// TIA Portal project "Al Qasim" (V16)

(* hardware
DEVICE "S7-1200 station_1"  S7-1200 Station
   slot 0: "Rack_0"  S7-1200 Rack  Rack  V1.0
   slot 1: "George"  CPU 1212C AC/DC/Rly  6ES7 212-1BE40-0XB0  V4.3
   slot 2: "DI 16x24VDC_1"  6ES7 221-1BF32-0XB0  V2.0
   slot 3: "CB 1241 (RS485)"  CB 1241 (RS485)  6ES7 241-1CH30-1XB0  V1.0
*)

// ===== PLC "George"  CPU 1212C AC/DC/Rly =====

VAR_GLOBAL   // PLC tag table "Default tag table"
   "System_Byte" AT %MB1000 : Byte;
   "FirstScan" AT %M1000.0 : Bool;
   "DiagStatusUpdate" AT %M1000.1 : Bool;
   "AlwaysTRUE" AT %M1000.2 : Bool;
   "AlwaysFALSE" AT %M1000.3 : Bool;
   "Clock_Byte" AT %MB1001 : Byte;
   "Clock_10Hz" AT %M1001.0 : Bool;
   "Clock_5Hz" AT %M1001.1 : Bool;
   "Clock_2.5Hz" AT %M1001.2 : Bool;
   "Clock_2Hz" AT %M1001.3 : Bool;
   "Clock_1.25Hz" AT %M1001.4 : Bool;
   "Clock_1Hz" AT %M1001.5 : Bool;
   "Clock_0.625Hz" AT %M1001.6 : Bool;
   "Clock_0.5Hz" AT %M1001.7 : Bool;
   "TS in Progress" AT %M0.0 : Bool;
   "TS Complete" AT %M0.1 : Bool;
   "initial switch ok" AT %M0.2 : Bool;
   "Datalog pulse" AT %M0.4 : Bool;
   "save name" AT %MB3 : Char;
   "allow datalogging" AT %M0.5 : Bool;
END_VAR

VAR_GLOBAL   // PLC tag table "Inputs"
   "Master Overide" AT %I0.0 : Bool;
   "Overide Pump 1" AT %I0.1 : Bool;
   "Overide Pump 2" AT %I0.2 : Bool;
   "Overide Pump 3" AT %I0.3 : Bool;
   "Overide Pump 4" AT %I0.4 : Bool;
   "Overide Pump 5" AT %I0.5 : Bool;
   "Float Inlet" AT %I0.6 : Bool;
   "Float Outlet" AT %I0.7 : Bool;
   "Float Stage" AT %I1.0 : Bool;
   "PB_Start" AT %I1.1 : Bool;
   "PB_Stop" AT %I1.2 : Bool;
END_VAR

VAR_GLOBAL   // PLC tag table "Outputs"
   "Pump 1" AT %Q0.0 : Bool;
   "Pump 2" AT %Q0.1 : Bool;
   "Pump 3" AT %Q0.2 : Bool;
   "Pump 4" AT %Q0.3 : Bool;
   "Pump 5" AT %Q0.4 : Bool;
   "Prog is running" AT %Q0.5 : Bool;
END_VAR

VAR_GLOBAL   // PLC tag table "Memory"
   "Main Function Loop" AT %MW1 : Int;   // 0= start up, 1 = stop, 2 = go, =3 Master Control
   "Run Mode" AT %MW4 : Int;   // 0 = Normal running, 1= tank switch, 2 inverted Humidity error
   "Tank Switch Mode Bit" AT %MW6 : Int;
   "OK to Switch" AT %M8.0 : Bool;
   "addy" AT %MW10 : Int;
   "Start a datalog session" AT %M0.3 : Bool;
   "logging ID" AT %MD12 : DInt;
   "OS log reset" AT %M0.6 : Bool;
   "OS1" AT %M0.7 : Bool;
END_VAR

VAR_GLOBAL   // PLC tag table "Retained memory"
   "Namer Logger" AT %MD1 : DInt;
   "name logger 2" AT %MD16 : DInt;
END_VAR

DATA_BLOCK "Stop_DB"   // DB1
{ S7_Optimized_Access := 'TRUE' }
VERSION : 0.1
// stored: InstanceOfName Stop
"Stop"
BEGIN
END_DATA_BLOCK

DATA_BLOCK "Auto Run_DB"   // DB2
{ S7_Optimized_Access := 'TRUE' }
VERSION : 0.1
// stored: InstanceOfName Auto Run
"Auto Run"
BEGIN
END_DATA_BLOCK

DATA_BLOCK "Manual Control_DB"   // DB9
{ S7_Optimized_Access := 'TRUE' }
VERSION : 0.1
// stored: InstanceOfName Manual Control
"Manual Control"
BEGIN
END_DATA_BLOCK

DATA_BLOCK "Modbus_DB"   // DB14
{ S7_Optimized_Access := 'TRUE' }
VERSION : 0.1
// stored: InstanceOfName Modbus
"Modbus"
BEGIN
END_DATA_BLOCK

DATA_BLOCK "Data process_DB"   // DB15
{ S7_Optimized_Access := 'TRUE' }
VERSION : 0.1
// stored: InstanceOfName Data process
"Data process"
BEGIN
END_DATA_BLOCK

// folder: Data

DATA_BLOCK "Data"   // DB3
{ S7_Optimized_Access := 'TRUE' }
VERSION : 0.1
   VAR
      "Inside Humidity" : Real := 80.0;
      "Inside Temp" : Real := 20.0;
      "Outside Humidity" : Real := 20.0;
      "Outside Temp" : Real := 30.0;
      "Temp Set Point" : Real := 18.0;
      "Hum Diff Set Point" : Real := 5.0;
      "Reset Timer" : Time := T#60s;
      "Tank Switch in progress" : Real;   // When Tank is switching, value is 100
      "Min Humidity" : Real := 40.0;   // Min humidity coming off the pad
   END_VAR
BEGIN
END_DATA_BLOCK

DATA_BLOCK "Modbus Data"   // DB13
{ S7_Optimized_Access := 'FALSE' }
VERSION : 0.1
   VAR
      "H&T" : Array[0..1] of Int;
      "Modbus Busy" : Bool;
   END_VAR
BEGIN
END_DATA_BLOCK

// folder: Data/Data Logging

DATA_BLOCK "Data Logging Config"   // DB21
{ S7_Optimized_Access := 'TRUE' }
VERSION : 0.1
   VAR
      "Name" : String := 'ash';
      ID : DInt := 0;
      Hedder : String := 'Ambient Temp,Ambient Hum,Inside Temp,Inside Hum,Tank Switch In Progress';
      "Data Log Data" : Struct
         "Data to be logged" : Array[0..4] of Real;
      END_STRUCT;
      "Start Done" : Bool;
      "Memory Allocation" : DInt := 5000;
      "Datalog Time Interval" : Time := T#1S;
   END_VAR
BEGIN
END_DATA_BLOCK

DATA_BLOCK "Create Data Log_DB"   // DB22
{ S7_Optimized_Access := 'TRUE' }
VERSION : 0.1
// stored: InstanceOfName Create Data Log
"Create Data Log"
BEGIN
END_DATA_BLOCK

// folder: Program Modes

DATA_BLOCK "Normal Running_DB"   // DB4
{ S7_Optimized_Access := 'TRUE' }
VERSION : 0.1
// stored: InstanceOfName Normal Running
"Normal Running"
BEGIN
END_DATA_BLOCK

DATA_BLOCK "Tank Switch_DB"   // DB5
{ S7_Optimized_Access := 'TRUE' }
VERSION : 0.1
// stored: InstanceOfName Tank Switch
"Tank Switch"
BEGIN
END_DATA_BLOCK

DATA_BLOCK "Tank Switch_DB_1"   // DB7
{ S7_Optimized_Access := 'TRUE' }
VERSION : 0.1
// stored: InstanceOfName Tank Switch
"Tank Switch"
BEGIN
END_DATA_BLOCK

DATA_BLOCK "Stop_DB_1"   // DB8
{ S7_Optimized_Access := 'TRUE' }
VERSION : 0.1
// stored: InstanceOfName Stop
"Stop"
BEGIN
END_DATA_BLOCK

DATA_BLOCK "Normal Running_DB_1"   // DB17
{ S7_Optimized_Access := 'TRUE' }
VERSION : 0.1
// stored: InstanceOfName Normal Running
"Normal Running"
BEGIN
END_DATA_BLOCK

DATA_BLOCK "Data Logging_DB"   // DB25
{ S7_Optimized_Access := 'TRUE' }
VERSION : 0.1
// stored: InstanceOfName Data Logging
"Data Logging"
BEGIN
END_DATA_BLOCK

// folder: System blocks/Program resources

DATA_BLOCK "IEC_Timer_0_DB"   // DB6
{ S7_Optimized_Access := 'TRUE' }
AUTHOR : Simatic
FAMILY : IEC
NAME : IEC_TMR
VERSION : 1.0
// stored: InstanceOfName IEC_TIMER
"IEC_TIMER"
BEGIN
END_DATA_BLOCK

DATA_BLOCK "IEC_Timer_0_DB_2"   // DB11
{ S7_Optimized_Access := 'TRUE' }
AUTHOR : Simatic
FAMILY : IEC
NAME : IEC_TMR
VERSION : 1.0
// stored: InstanceOfName IEC_TIMER
"IEC_TIMER"
BEGIN
END_DATA_BLOCK

DATA_BLOCK "IEC_Timer_0_DB_3"   // DB16
{ S7_Optimized_Access := 'TRUE' }
AUTHOR : Simatic
FAMILY : IEC
NAME : IEC_TMR
VERSION : 1.0
// stored: InstanceOfName IEC_TIMER
"IEC_TIMER"
BEGIN
END_DATA_BLOCK

DATA_BLOCK "IEC_Timer_0_DB_1"   // DB24
{ S7_Optimized_Access := 'TRUE' }
AUTHOR : Simatic
FAMILY : IEC
NAME : IEC_TMR
VERSION : 1.0
// stored: InstanceOfName IEC_TIMER
"IEC_TIMER"
BEGIN
END_DATA_BLOCK

// folder: (top level)

FUNCTION_BLOCK "Modbus"   // FB6, LAD
{ S7_Optimized_Access := 'TRUE' }
VERSION : 0.1
BEGIN

REGION Network 1: To read T&H from 2 sensors @ address 2 and 3
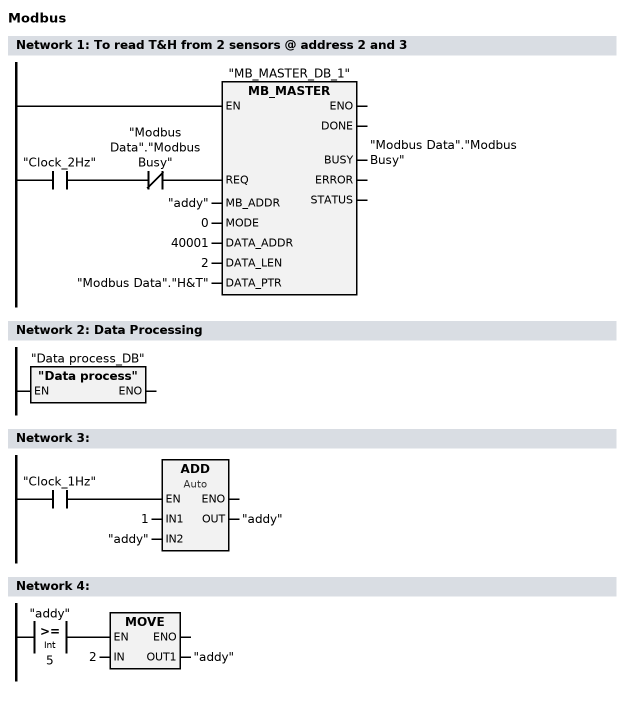
   "MB_MASTER_DB_1"(REQ := "Clock_2Hz" AND NOT "Modbus Data"."Modbus Busy",   // MB_MASTER
                    MB_ADDR := "addy",
                    MODE := 0,
                    DATA_ADDR := 40001,
                    DATA_LEN := 2,
                    DATA_PTR := "Modbus Data"."H&T",
                    BUSY => "Modbus Data"."Modbus Busy");
END_REGION

REGION Network 2: Data Processing
   RUNG wire#powerrail
      "Data process_DB"()
   END_RUNG
   // the same network as SCL:
   "Data process_DB"();   // "Data process"
END_REGION

REGION Network 3
   RUNG wire#powerrail
      Contact( "Clock_1Hz" )
      Add(in1 := 1, in2 := "addy", out => "addy")
   END_RUNG
   // the same network as SCL:
   IF "Clock_1Hz" THEN "addy" := 1 + "addy"; END_IF;
END_REGION

REGION Network 4
   RUNG wire#powerrail
      { S7_Templates := "SrcType := Int" } GE_Contact(in1 := "addy", in2 := 5)
      Move(in := 2, out1 => "addy")
   END_RUNG
   // the same network as SCL:
   IF "addy" >= 5 THEN "addy" := 2; END_IF;
END_REGION
END_FUNCTION_BLOCK

ORGANIZATION_BLOCK "Main"   // OB1, LAD, ProgramCycle
TITLE = "Main Program Sweep (Cycle)"
{ S7_Optimized_Access := 'TRUE' }
VERSION : 0.1
   VAR_INPUT
      Initial_Call : Bool;   // Initial call of this OB
      Remanence : Bool;   // =True, if remanent data are available
   END_VAR
   VAR_TEMP   // added for the SCL form of the ladder/FBD networks
      _w1 : Bool;
      _w2 : Bool;
   END_VAR
BEGIN

REGION Network 1: Select Main function Loop
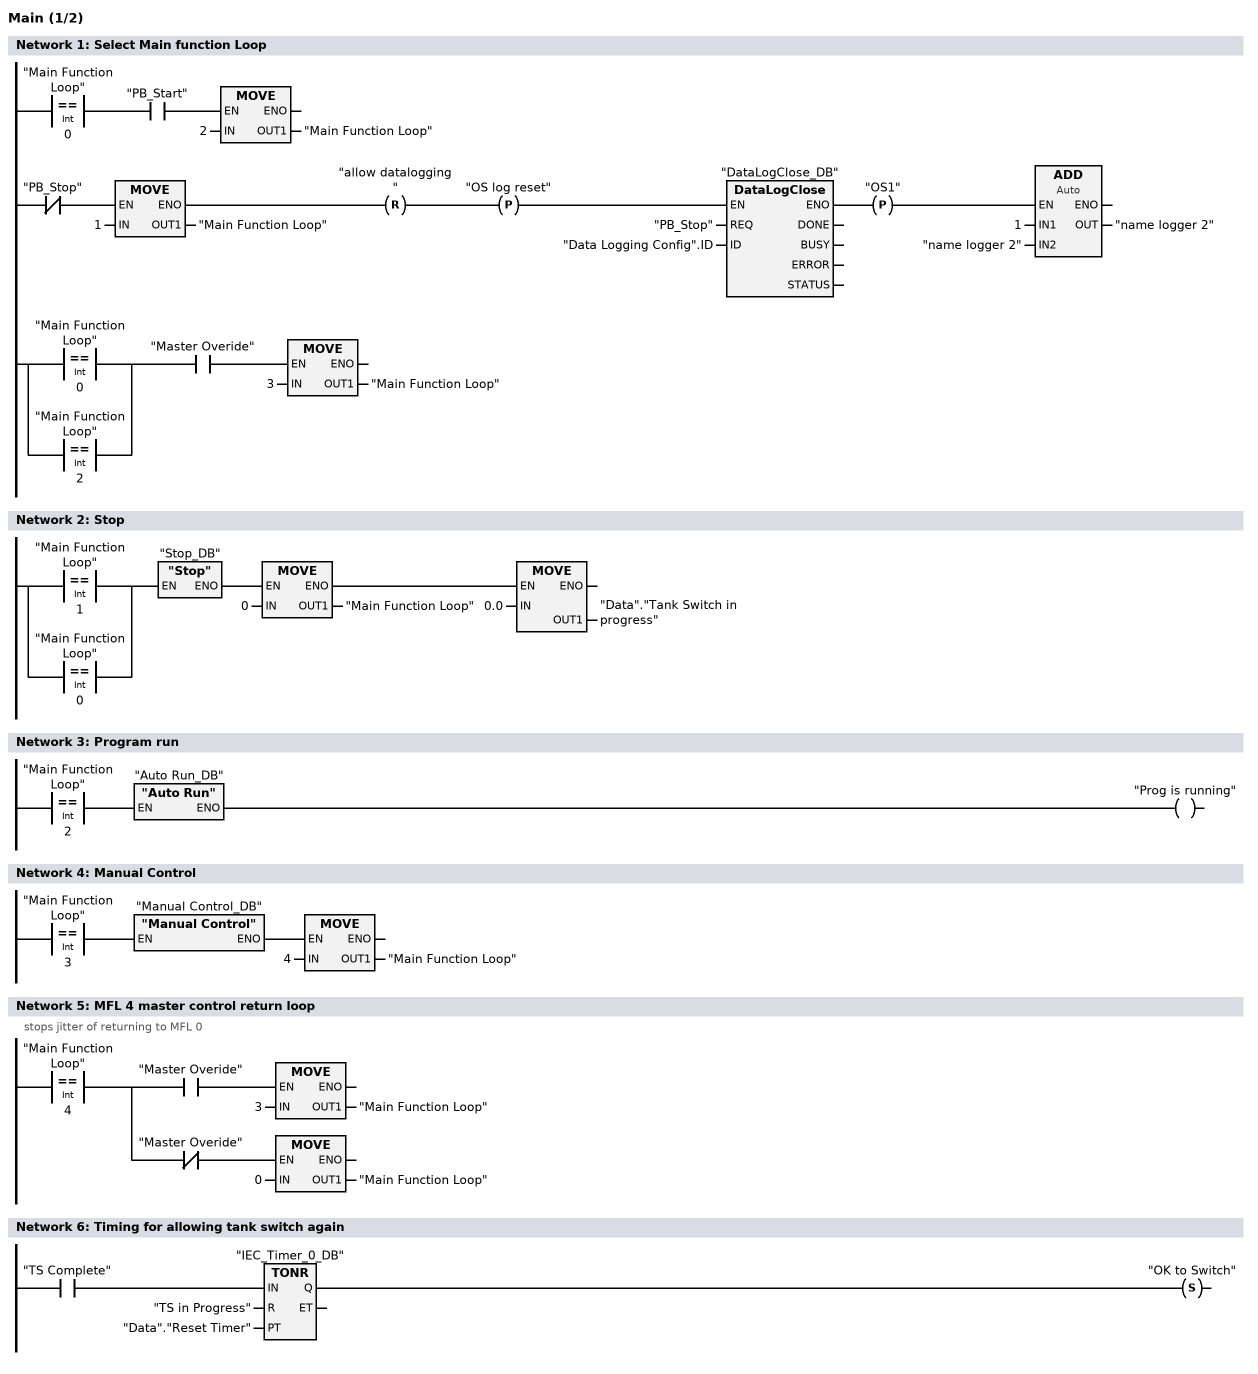
   // ENO of a box is taken as its EN; it also drops when the box reports an error
   IF ("Main Function Loop" = 0) AND "PB_Start" THEN "Main Function Loop" := 2; END_IF;
   IF NOT "PB_Stop" THEN
       "Main Function Loop" := 1;
       "allow datalogging" := FALSE;
   END_IF;
   #_w1 := NOT "PB_Stop" AND NOT "OS log reset";   // rising edge
   "OS log reset" := NOT "PB_Stop";
   IF #_w1 THEN
       "DataLogClose_DB"(REQ := "PB_Stop", ID := "Data Logging Config".ID);   // DataLogClose
   END_IF;
   #_w2 := #_w1 AND NOT "OS1";   // rising edge
   "OS1" := #_w1;
   IF #_w2 THEN "name logger 2" := 1 + "name logger 2"; END_IF;
   IF (("Main Function Loop" = 0) OR ("Main Function Loop" = 2)) AND "Master Overide" THEN
       "Main Function Loop" := 3;
   END_IF;
END_REGION

REGION Network 2: Stop
   RUNG wire#powerrail
      { S7_Templates := "SrcType := Int" } EQ_Contact(in1 := "Main Function Loop", in2 := 1)
      wire#w1
      "Stop_DB"()
      Move(in := 0, out1 => "Main Function Loop")
      Move(in := 0.0, out1 => "Data"."Tank Switch in progress")
   END_RUNG
   RUNG wire#powerrail
      { S7_Templates := "SrcType := Int" } EQ_Contact(in1 := "Main Function Loop", in2 := 0)
   END_RUNG wire#w1
   // the same network as SCL:
   "Stop_DB"(EN := ("Main Function Loop" = 1) OR ("Main Function Loop" = 0), ENO => #_w1);   // "Stop"
   IF #_w1 THEN
       "Main Function Loop" := 0;
       "Data"."Tank Switch in progress" := 0.0;
   END_IF;
END_REGION

REGION Network 3: Program run
   RUNG wire#powerrail
      { S7_Templates := "SrcType := Int" } EQ_Contact(in1 := "Main Function Loop", in2 := 2)
      "Auto Run_DB"()
      Coil( "Prog is running" )
   END_RUNG
   // the same network as SCL:
   "Auto Run_DB"(EN := "Main Function Loop" = 2, ENO => #_w1);   // "Auto Run"
   "Prog is running" := #_w1;
END_REGION

REGION Network 4: Manual Control
   RUNG wire#powerrail
      { S7_Templates := "SrcType := Int" } EQ_Contact(in1 := "Main Function Loop", in2 := 3)
      "Manual Control_DB"()
      Move(in := 4, out1 => "Main Function Loop")
   END_RUNG
   // the same network as SCL:
   "Manual Control_DB"(EN := "Main Function Loop" = 3, ENO => #_w1);   // "Manual Control"
   IF #_w1 THEN "Main Function Loop" := 4; END_IF;
END_REGION

REGION Network 5: MFL 4 master control return loop
   // stops jitter of returning to MFL 0
   RUNG wire#powerrail
      { S7_Templates := "SrcType := Int" } EQ_Contact(in1 := "Main Function Loop", in2 := 4)
      wire#w1
      Contact( "Master Overide" )
      Move(in := 3, out1 => "Main Function Loop")
   END_RUNG
   RUNG wire#w1
      I_Contact( "Master Overide" )
      Move(in := 0, out1 => "Main Function Loop")
   END_RUNG
   // the same network as SCL:
   #_w1 := "Main Function Loop" = 4;
   IF #_w1 AND "Master Overide" THEN "Main Function Loop" := 3; END_IF;
   IF #_w1 AND NOT "Master Overide" THEN "Main Function Loop" := 0; END_IF;
END_REGION

REGION Network 6: Timing for allowing tank switch again
   "IEC_Timer_0_DB".TONR(IN := "TS Complete", R := "TS in Progress", PT := "Data"."Reset Timer");
   IF "IEC_Timer_0_DB".Q THEN "OK to Switch" := TRUE; END_IF;
END_REGION

REGION Network 7: reset easter egg (hold stop for 5 sec)
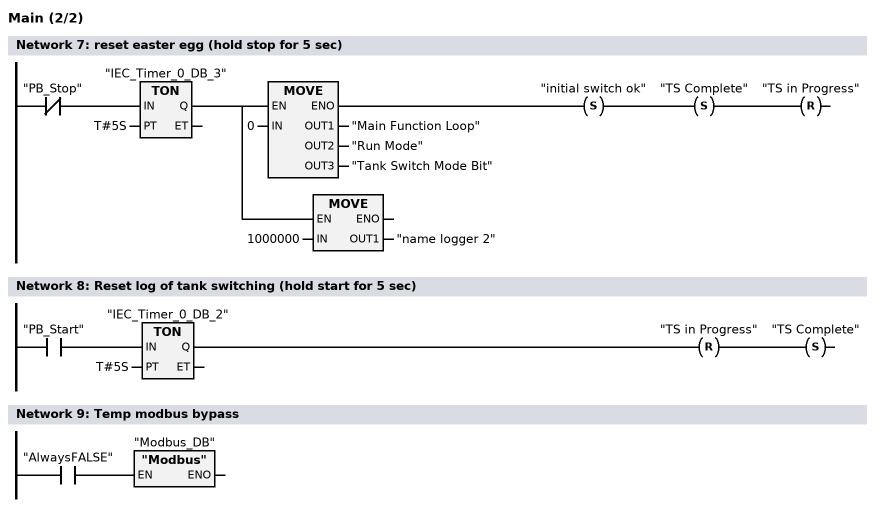
   "IEC_Timer_0_DB_3".TON(IN := NOT "PB_Stop", PT := T#5S);
   IF "IEC_Timer_0_DB_3".Q THEN
       "Main Function Loop" := 0;
       "Run Mode" := 0;
       "Tank Switch Mode Bit" := 0;
       "initial switch ok" := TRUE;
       "TS Complete" := TRUE;
       "TS in Progress" := FALSE;
       "name logger 2" := 1000000;
   END_IF;
END_REGION

REGION Network 8: Reset log of tank switching (hold start for 5 sec)
   "IEC_Timer_0_DB_2".TON(IN := "PB_Start", PT := T#5S);
   IF "IEC_Timer_0_DB_2".Q THEN
       "TS in Progress" := FALSE;
       "TS Complete" := TRUE;
   END_IF;
END_REGION

REGION Network 9: Temp modbus bypass
   RUNG wire#powerrail
      Contact( "AlwaysFALSE" )
      "Modbus_DB"()
   END_RUNG
   // the same network as SCL:
   IF "AlwaysFALSE" THEN
       "Modbus_DB"();   // "Modbus"
   END_IF;
END_REGION
END_ORGANIZATION_BLOCK

ORGANIZATION_BLOCK "Startup"   // OB100, LAD, Startup
TITLE = "Complete Restart"
{ S7_Optimized_Access := 'TRUE' }
VERSION : 0.1
   VAR_INPUT
      LostRetentive : Bool;   // True if retentive data are lost
      LostRTC : Bool;   // True if date and time are lost
   END_VAR
BEGIN

REGION Network 1
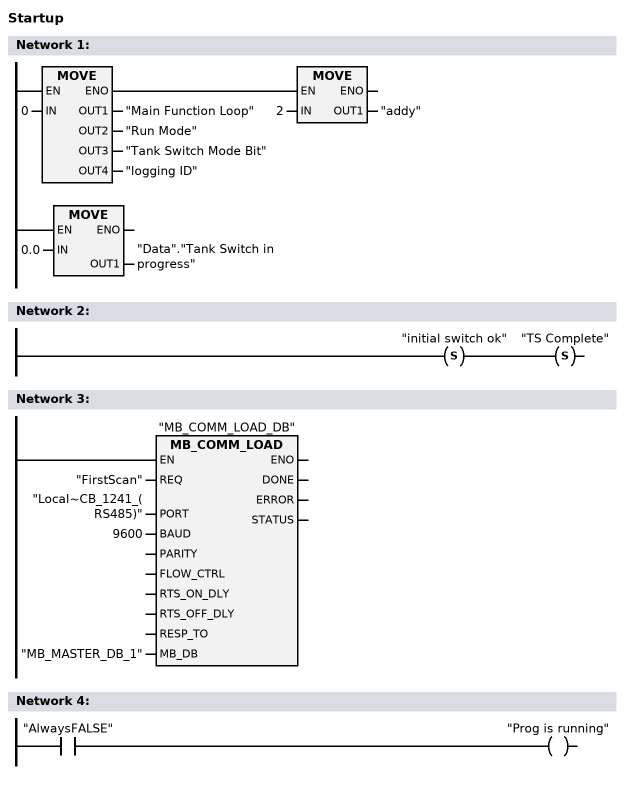
   RUNG wire#powerrail
      Move(in := 0, out1 => "Main Function Loop", out2 => "Run Mode", out3 => "Tank Switch Mode Bit", out4 => "logging ID")
      Move(in := 2, out1 => "addy")
   END_RUNG
   RUNG wire#powerrail
      Move(in := 0.0, out1 => "Data"."Tank Switch in progress")
   END_RUNG
   // the same network as SCL:
   "Main Function Loop" := 0;
   "Run Mode" := 0;
   "Tank Switch Mode Bit" := 0;
   "logging ID" := 0;
   "addy" := 2;
   "Data"."Tank Switch in progress" := 0.0;
END_REGION

REGION Network 2
   RUNG wire#powerrail
      S_Coil( "initial switch ok" )
      S_Coil( "TS Complete" )
   END_RUNG
   // the same network as SCL:
   "initial switch ok" := TRUE;
   "TS Complete" := TRUE;
END_REGION

REGION Network 3
   "MB_COMM_LOAD_DB"(REQ := "FirstScan",   // MB_COMM_LOAD
                     PORT := "Local~CB_1241_(RS485)",
                     BAUD := 9600,
                     MB_DB := "MB_MASTER_DB_1");
END_REGION

REGION Network 4
   RUNG wire#powerrail
      Contact( "AlwaysFALSE" )
      Coil( "Prog is running" )
   END_RUNG
   // the same network as SCL:
   "Prog is running" := "AlwaysFALSE";
END_REGION
END_ORGANIZATION_BLOCK

// folder: Data

FUNCTION_BLOCK "Data process"   // FB7, LAD
{ S7_Optimized_Access := 'TRUE' }
VERSION : 0.1
   VAR
      "hum tempo" : Int;
   END_VAR
   VAR_TEMP
      "temp tempo" : Int;
   END_VAR
BEGIN

REGION Network 1: Inside Sensor
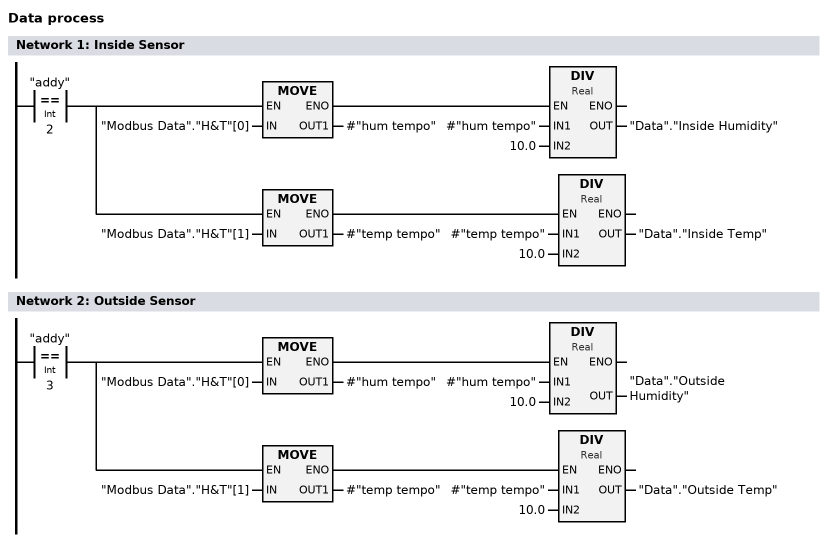
   RUNG wire#powerrail
      { S7_Templates := "SrcType := Int" } EQ_Contact(in1 := "addy", in2 := 2)
      wire#w1
      Move(in := "Modbus Data"."H&T"[0], out1 => #"hum tempo")
      { S7_Templates := "SrcType := Real" } Div(in1 := #"hum tempo", in2 := 10.0, out => "Data"."Inside Humidity")
   END_RUNG
   RUNG wire#w1
      Move(in := "Modbus Data"."H&T"[1], out1 => #"temp tempo")
      { S7_Templates := "SrcType := Real" } Div(in1 := #"temp tempo", in2 := 10.0, out => "Data"."Inside Temp")
   END_RUNG
   // the same network as SCL:
   IF "addy" = 2 THEN
       #"hum tempo" := "Modbus Data"."H&T"[0];
       "Data"."Inside Humidity" := #"hum tempo" / 10.0;
       #"temp tempo" := "Modbus Data"."H&T"[1];
       "Data"."Inside Temp" := #"temp tempo" / 10.0;
   END_IF;
END_REGION

REGION Network 2: Outside Sensor
   RUNG wire#powerrail
      { S7_Templates := "SrcType := Int" } EQ_Contact(in1 := "addy", in2 := 3)
      wire#w1
      Move(in := "Modbus Data"."H&T"[0], out1 => #"hum tempo")
      { S7_Templates := "SrcType := Real" } Div(in1 := #"hum tempo", in2 := 10.0, out => "Data"."Outside Humidity")
   END_RUNG
   RUNG wire#w1
      Move(in := "Modbus Data"."H&T"[1], out1 => #"temp tempo")
      { S7_Templates := "SrcType := Real" } Div(in1 := #"temp tempo", in2 := 10.0, out => "Data"."Outside Temp")
   END_RUNG
   // the same network as SCL:
   IF "addy" = 3 THEN
       #"hum tempo" := "Modbus Data"."H&T"[0];
       "Data"."Outside Humidity" := #"hum tempo" / 10.0;
       #"temp tempo" := "Modbus Data"."H&T"[1];
       "Data"."Outside Temp" := #"temp tempo" / 10.0;
   END_IF;
END_REGION
END_FUNCTION_BLOCK

// folder: Data/Data Logging

FUNCTION_BLOCK "Data Logging"   // FB8, LAD
{ S7_Optimized_Access := 'TRUE' }
VERSION : 0.1
   VAR
      "OS Datalog" : Bool;
      "pulse reset" : Bool;
   END_VAR
BEGIN

REGION Network 1: when Datalogging is run, start a new session by creating a data log
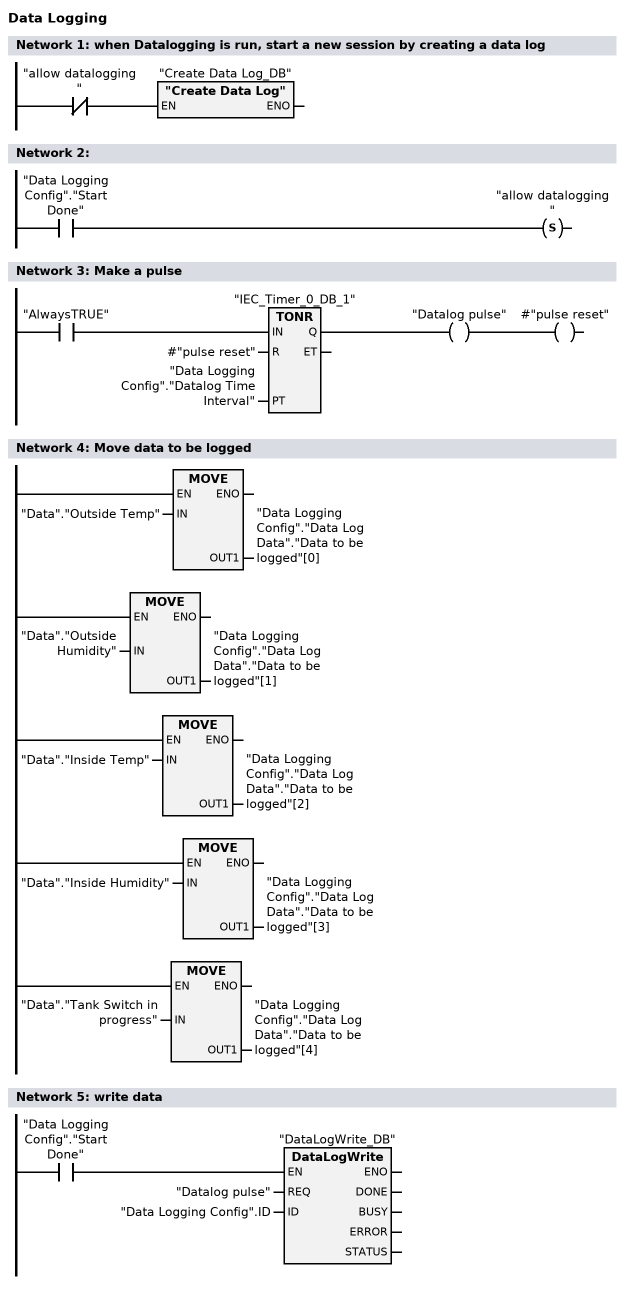
   RUNG wire#powerrail
      I_Contact( "allow datalogging" )
      "Create Data Log_DB"()
   END_RUNG
   // the same network as SCL:
   IF NOT "allow datalogging" THEN
       "Create Data Log_DB"();   // "Create Data Log"
   END_IF;
END_REGION

REGION Network 2
   RUNG wire#powerrail
      Contact( "Data Logging Config"."Start Done" )
      S_Coil( "allow datalogging" )
   END_RUNG
   // the same network as SCL:
   IF "Data Logging Config"."Start Done" THEN "allow datalogging" := TRUE; END_IF;
END_REGION

REGION Network 3: Make a pulse
   "IEC_Timer_0_DB_1".TONR(IN := "AlwaysTRUE",
                           R := #"pulse reset",
                           PT := "Data Logging Config"."Datalog Time Interval");
   "Datalog pulse" := "IEC_Timer_0_DB_1".Q;
   #"pulse reset" := "IEC_Timer_0_DB_1".Q;
END_REGION

REGION Network 4: Move data to be logged
   RUNG wire#powerrail
      Move(in := "Data"."Outside Temp", out1 => "Data Logging Config"."Data Log Data"."Data to be logged"[0])
   END_RUNG
   RUNG wire#powerrail
      Move(in := "Data"."Outside Humidity", out1 => "Data Logging Config"."Data Log Data"."Data to be logged"[1])
   END_RUNG
   RUNG wire#powerrail
      Move(in := "Data"."Inside Temp", out1 => "Data Logging Config"."Data Log Data"."Data to be logged"[2])
   END_RUNG
   RUNG wire#powerrail
      Move(in := "Data"."Inside Humidity", out1 => "Data Logging Config"."Data Log Data"."Data to be logged"[3])
   END_RUNG
   RUNG wire#powerrail
      Move(in := "Data"."Tank Switch in progress", out1 => "Data Logging Config"."Data Log Data"."Data to be logged"[4])
   END_RUNG
   // the same network as SCL:
   "Data Logging Config"."Data Log Data"."Data to be logged"[0] := "Data"."Outside Temp";
   "Data Logging Config"."Data Log Data"."Data to be logged"[1] := "Data"."Outside Humidity";
   "Data Logging Config"."Data Log Data"."Data to be logged"[2] := "Data"."Inside Temp";
   "Data Logging Config"."Data Log Data"."Data to be logged"[3] := "Data"."Inside Humidity";
   "Data Logging Config"."Data Log Data"."Data to be logged"[4] := "Data"."Tank Switch in progress";
END_REGION

REGION Network 5: write data
   IF "Data Logging Config"."Start Done" THEN
       "DataLogWrite_DB"(REQ := "Datalog pulse", ID := "Data Logging Config".ID);   // DataLogWrite
   END_IF;
END_REGION
END_FUNCTION_BLOCK

FUNCTION_BLOCK "Create Data Log"   // FB9, LAD
{ S7_Optimized_Access := 'TRUE' }
VERSION : 0.1
   VAR
      "OS logging" : Bool;
   END_VAR
   VAR_TEMP
      test : WChar;
      tbf : String;
   END_VAR
BEGIN

REGION Network 1: Create name
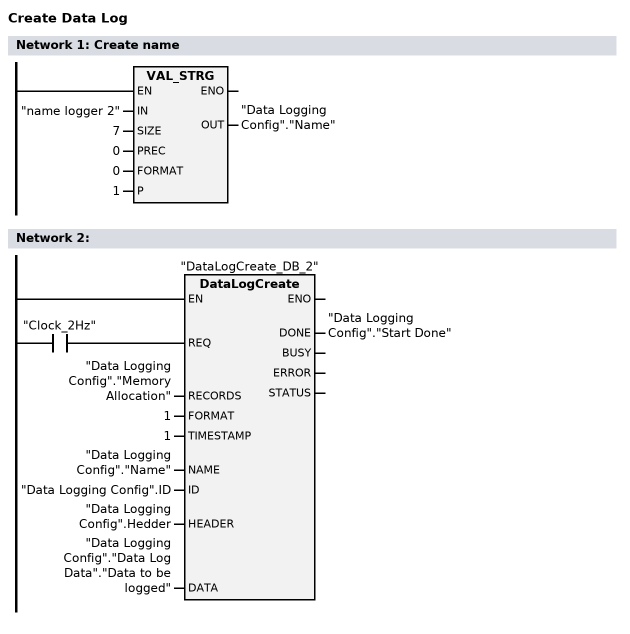
   VAL_STRG(IN := "name logger 2",
            SIZE := 7,
            PREC := 0,
            FORMAT := 0,
            P := 1,
            OUT => "Data Logging Config"."Name");
END_REGION

REGION Network 2
   "DataLogCreate_DB_2"(REQ := "Clock_2Hz",   // DataLogCreate
                        RECORDS := "Data Logging Config"."Memory Allocation",
                        FORMAT := 1,
                        TIMESTAMP := 1,
                        "NAME" := "Data Logging Config"."Name",
                        ID := "Data Logging Config".ID,
                        HEADER := "Data Logging Config".Hedder,
                        DATA := "Data Logging Config"."Data Log Data"."Data to be logged",
                        DONE => "Data Logging Config"."Start Done");
END_REGION
END_FUNCTION_BLOCK

// folder: Program Modes

FUNCTION_BLOCK "Stop"   // FB1, LAD
{ S7_Optimized_Access := 'TRUE' }
VERSION : 0.1
BEGIN

REGION Network 1
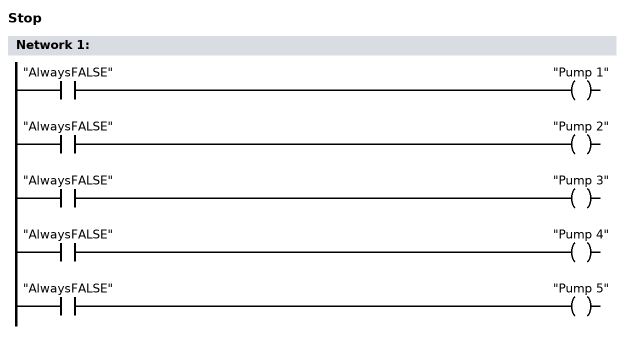
   RUNG wire#powerrail
      Contact( "AlwaysFALSE" )
      Coil( "Pump 1" )
   END_RUNG
   RUNG wire#powerrail
      Contact( "AlwaysFALSE" )
      Coil( "Pump 2" )
   END_RUNG
   RUNG wire#powerrail
      Contact( "AlwaysFALSE" )
      Coil( "Pump 3" )
   END_RUNG
   RUNG wire#powerrail
      Contact( "AlwaysFALSE" )
      Coil( "Pump 4" )
   END_RUNG
   RUNG wire#powerrail
      Contact( "AlwaysFALSE" )
      Coil( "Pump 5" )
   END_RUNG
   // the same network as SCL:
   "Pump 1" := "AlwaysFALSE";
   "Pump 2" := "AlwaysFALSE";
   "Pump 3" := "AlwaysFALSE";
   "Pump 4" := "AlwaysFALSE";
   "Pump 5" := "AlwaysFALSE";
END_REGION
END_FUNCTION_BLOCK

FUNCTION_BLOCK "Tank Switch"   // FB2, LAD
{ S7_Optimized_Access := 'TRUE' }
VERSION : 0.1
   VAR_TEMP   // added for the SCL form of the ladder/FBD networks
      _w1 : Bool;
   END_VAR
BEGIN

REGION Network 1
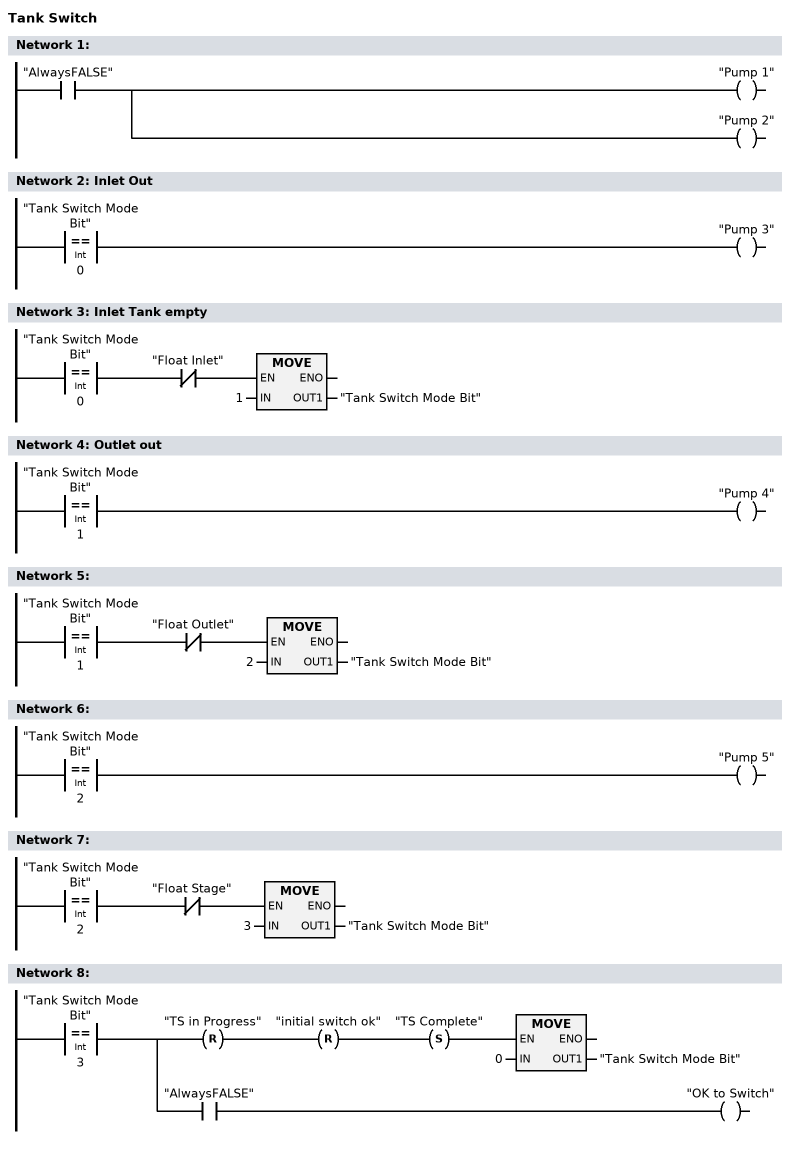
   RUNG wire#powerrail
      Contact( "AlwaysFALSE" )
      wire#w1
      Coil( "Pump 1" )
   END_RUNG
   RUNG wire#w1
      Coil( "Pump 2" )
   END_RUNG
   // the same network as SCL:
   "Pump 1" := "AlwaysFALSE";
   "Pump 2" := "AlwaysFALSE";
END_REGION

REGION Network 2: Inlet Out
   RUNG wire#powerrail
      { S7_Templates := "SrcType := Int" } EQ_Contact(in1 := "Tank Switch Mode Bit", in2 := 0)
      Coil( "Pump 3" )
   END_RUNG
   // the same network as SCL:
   "Pump 3" := "Tank Switch Mode Bit" = 0;
END_REGION

REGION Network 3: Inlet Tank empty
   RUNG wire#powerrail
      { S7_Templates := "SrcType := Int" } EQ_Contact(in1 := "Tank Switch Mode Bit", in2 := 0)
      I_Contact( "Float Inlet" )
      Move(in := 1, out1 => "Tank Switch Mode Bit")
   END_RUNG
   // the same network as SCL:
   IF ("Tank Switch Mode Bit" = 0) AND NOT "Float Inlet" THEN "Tank Switch Mode Bit" := 1; END_IF;
END_REGION

REGION Network 4: Outlet out
   RUNG wire#powerrail
      { S7_Templates := "SrcType := Int" } EQ_Contact(in1 := "Tank Switch Mode Bit", in2 := 1)
      Coil( "Pump 4" )
   END_RUNG
   // the same network as SCL:
   "Pump 4" := "Tank Switch Mode Bit" = 1;
END_REGION

REGION Network 5
   RUNG wire#powerrail
      { S7_Templates := "SrcType := Int" } EQ_Contact(in1 := "Tank Switch Mode Bit", in2 := 1)
      I_Contact( "Float Outlet" )
      Move(in := 2, out1 => "Tank Switch Mode Bit")
   END_RUNG
   // the same network as SCL:
   IF ("Tank Switch Mode Bit" = 1) AND NOT "Float Outlet" THEN "Tank Switch Mode Bit" := 2; END_IF;
END_REGION

REGION Network 6
   RUNG wire#powerrail
      { S7_Templates := "SrcType := Int" } EQ_Contact(in1 := "Tank Switch Mode Bit", in2 := 2)
      Coil( "Pump 5" )
   END_RUNG
   // the same network as SCL:
   "Pump 5" := "Tank Switch Mode Bit" = 2;
END_REGION

REGION Network 7
   RUNG wire#powerrail
      { S7_Templates := "SrcType := Int" } EQ_Contact(in1 := "Tank Switch Mode Bit", in2 := 2)
      I_Contact( "Float Stage" )
      Move(in := 3, out1 => "Tank Switch Mode Bit")
   END_RUNG
   // the same network as SCL:
   IF ("Tank Switch Mode Bit" = 2) AND NOT "Float Stage" THEN "Tank Switch Mode Bit" := 3; END_IF;
END_REGION

REGION Network 8
   RUNG wire#powerrail
      { S7_Templates := "SrcType := Int" } EQ_Contact(in1 := "Tank Switch Mode Bit", in2 := 3)
      wire#w1
      R_Coil( "TS in Progress" )
      R_Coil( "initial switch ok" )
      S_Coil( "TS Complete" )
      Move(in := 0, out1 => "Tank Switch Mode Bit")
   END_RUNG
   RUNG wire#w1
      Contact( "AlwaysFALSE" )
      Coil( "OK to Switch" )
   END_RUNG
   // the same network as SCL:
   #_w1 := "Tank Switch Mode Bit" = 3;
   IF #_w1 THEN
       "TS in Progress" := FALSE;
       "initial switch ok" := FALSE;
       "TS Complete" := TRUE;
       "Tank Switch Mode Bit" := 0;
   END_IF;
   "OK to Switch" := #_w1 AND "AlwaysFALSE";
END_REGION
END_FUNCTION_BLOCK

FUNCTION_BLOCK "Normal Running"   // FB3, LAD
{ S7_Optimized_Access := 'TRUE' }
VERSION : 0.1
BEGIN

REGION Network 1: Cooling pumps on
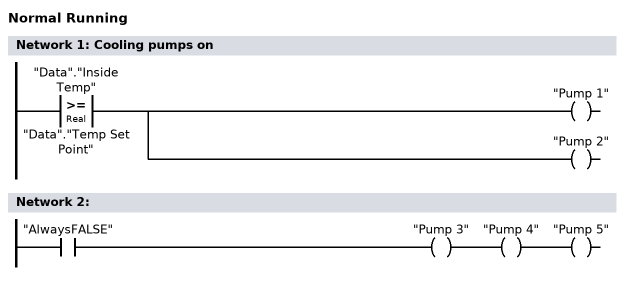
   RUNG wire#powerrail
      { S7_Templates := "SrcType := Real" } GE_Contact(in1 := "Data"."Inside Temp", in2 := "Data"."Temp Set Point")
      wire#w1
      Coil( "Pump 1" )
   END_RUNG
   RUNG wire#w1
      Coil( "Pump 2" )
   END_RUNG
   // the same network as SCL:
   "Pump 1" := "Data"."Inside Temp" >= "Data"."Temp Set Point";
   "Pump 2" := "Pump 1";
END_REGION

REGION Network 2
   RUNG wire#powerrail
      Contact( "AlwaysFALSE" )
      Coil( "Pump 3" )
      Coil( "Pump 4" )
      Coil( "Pump 5" )
   END_RUNG
   // the same network as SCL:
   "Pump 3" := "AlwaysFALSE";
   "Pump 4" := "AlwaysFALSE";
   "Pump 5" := "AlwaysFALSE";
END_REGION
END_FUNCTION_BLOCK

FUNCTION_BLOCK "Auto Run"   // FB4, LAD
{ S7_Optimized_Access := 'TRUE' }
VERSION : 0.1
   VAR
      OS1 : Bool;   // OS for setting tank switch latch
   END_VAR
   VAR_TEMP
      humdif : Real;
   END_VAR
   VAR_TEMP   // added for the SCL form of the ladder/FBD networks
      _w1 : Bool;
      _w2 : Bool;
   END_VAR
BEGIN

REGION Network 1: Calculate humidity difference
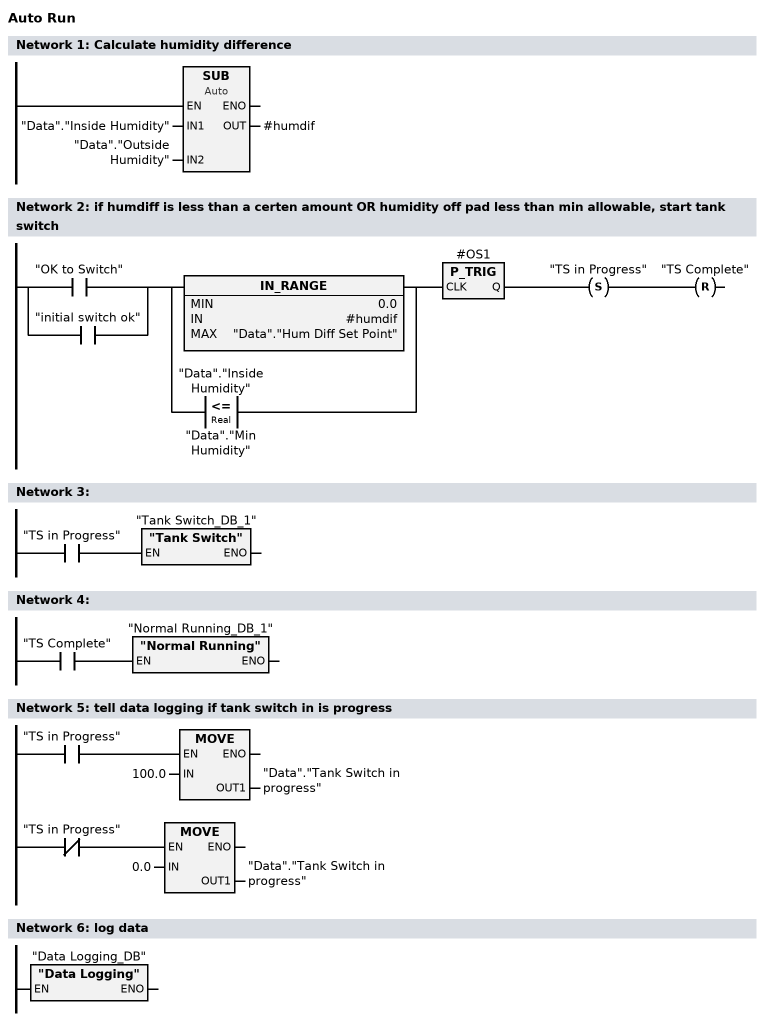
   RUNG wire#powerrail
      Sub(in1 := "Data"."Inside Humidity", in2 := "Data"."Outside Humidity", out => #humdif)
   END_RUNG
   // the same network as SCL:
   #humdif := "Data"."Inside Humidity" - "Data"."Outside Humidity";
END_REGION

REGION Network 2: if humdiff is less than a certen amount OR humidity off pad less than min allowable, start tank switch
   RUNG wire#powerrail
      Contact( "OK to Switch" )
      wire#w1
      { S7_Templates := "SrcType := Real" } InRange(min := 0.0, in := #humdif, max := "Data"."Hum Diff Set Point")
      wire#w2
      P_Trig( #OS1 )
      S_Coil( "TS in Progress" )
      R_Coil( "TS Complete" )
   END_RUNG
   RUNG wire#powerrail
      Contact( "initial switch ok" )
   END_RUNG wire#w1
   RUNG wire#w1
      { S7_Templates := "SrcType := Real" } LE_Contact(in1 := "Data"."Inside Humidity", in2 := "Data"."Min Humidity")
   END_RUNG wire#w2
   // the same network as SCL:
   #_w1 := ("OK to Switch" OR "initial switch ok") AND (((0.0 <= #humdif) AND (#humdif <= "Data"."Hum Diff Set Point")) OR ("Data"."Inside Humidity" <= "Data"."Min Humidity"));
   #_w2 := #_w1 AND NOT #OS1;   // rising edge
   #OS1 := #_w1;
   IF #_w2 THEN
       "TS in Progress" := TRUE;
       "TS Complete" := FALSE;
   END_IF;
END_REGION

REGION Network 3
   RUNG wire#powerrail
      Contact( "TS in Progress" )
      "Tank Switch_DB_1"()
   END_RUNG
   // the same network as SCL:
   IF "TS in Progress" THEN
       "Tank Switch_DB_1"();   // "Tank Switch"
   END_IF;
END_REGION

REGION Network 4
   RUNG wire#powerrail
      Contact( "TS Complete" )
      "Normal Running_DB_1"()
   END_RUNG
   // the same network as SCL:
   IF "TS Complete" THEN
       "Normal Running_DB_1"();   // "Normal Running"
   END_IF;
END_REGION

REGION Network 5: tell data logging if tank switch in is progress
   RUNG wire#powerrail
      Contact( "TS in Progress" )
      Move(in := 100.0, out1 => "Data"."Tank Switch in progress")
   END_RUNG
   RUNG wire#powerrail
      I_Contact( "TS in Progress" )
      Move(in := 0.0, out1 => "Data"."Tank Switch in progress")
   END_RUNG
   // the same network as SCL:
   IF "TS in Progress" THEN "Data"."Tank Switch in progress" := 100.0; END_IF;
   IF NOT "TS in Progress" THEN "Data"."Tank Switch in progress" := 0.0; END_IF;
END_REGION

REGION Network 6: log data
   RUNG wire#powerrail
      "Data Logging_DB"()
   END_RUNG
   // the same network as SCL:
   "Data Logging_DB"();   // "Data Logging"
END_REGION
END_FUNCTION_BLOCK

FUNCTION_BLOCK "Manual Control"   // FB5, LAD
{ S7_Optimized_Access := 'TRUE' }
VERSION : 0.1
BEGIN

REGION Network 1
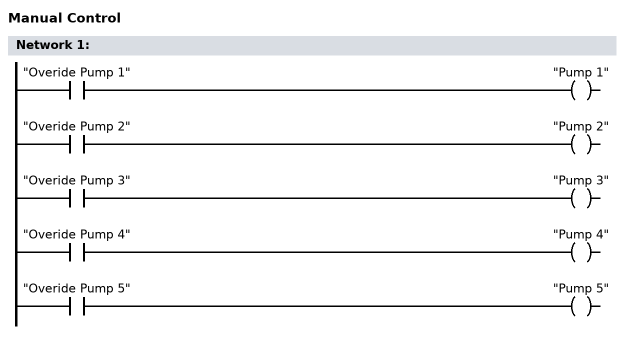
   RUNG wire#powerrail
      Contact( "Overide Pump 1" )
      Coil( "Pump 1" )
   END_RUNG
   RUNG wire#powerrail
      Contact( "Overide Pump 2" )
      Coil( "Pump 2" )
   END_RUNG
   RUNG wire#powerrail
      Contact( "Overide Pump 3" )
      Coil( "Pump 3" )
   END_RUNG
   RUNG wire#powerrail
      Contact( "Overide Pump 4" )
      Coil( "Pump 4" )
   END_RUNG
   RUNG wire#powerrail
      Contact( "Overide Pump 5" )
      Coil( "Pump 5" )
   END_RUNG
   // the same network as SCL:
   "Pump 1" := "Overide Pump 1";
   "Pump 2" := "Overide Pump 2";
   "Pump 3" := "Overide Pump 3";
   "Pump 4" := "Overide Pump 4";
   "Pump 5" := "Overide Pump 5";
END_REGION
END_FUNCTION_BLOCK